TYPE StepperPOSControl :
STRUCT
	Execute : BOOL;
	EmergencyStop : BOOL;
	TargetPosition : UDINT;
	Velocity : INT;
	StartType : UINT;
	Acceleration : UINT;
	Deceleration : UINT;
END_STRUCT
END_TYPE

(* stored: Version 1.1.0.1, ProductVersion 3.1.4024.11
   DUT StepperPOSControl: Id {87711e8a-4859-414c-902f-1710864272c2} *)
